FUNCTION_BLOCK SINGLE_EVENT_CONTROLLER (* Composite Function Block Type *)
  (* Standard: 61499-2 *)
  (* Version 1.0, 2019-03-16, adeel *)
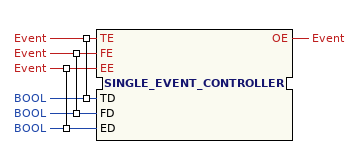
  EVENT_INPUT
    TE WITH TD; (* Initialization Request *)
    FE WITH FD; (* Normal Execution Request *)
    EE WITH ED;
  END_EVENT
  EVENT_OUTPUT
    OE; (* Initialization Confirm *)
  END_EVENT
  VAR_INPUT
    TD : BOOL; (* Input event qualifier *)
    FD : BOOL;
    ED : BOOL;
  END_VAR
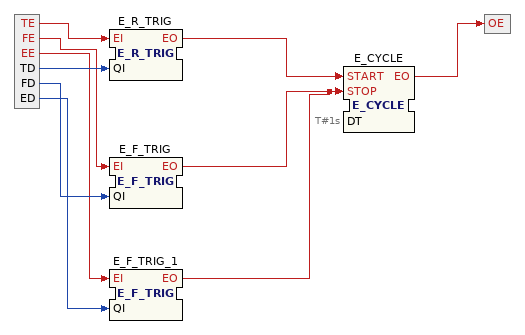
  FBS
    E_CYCLE : E_CYCLE(DT := T#1s);
    E_R_TRIG : E_R_TRIG;
    E_F_TRIG : E_F_TRIG;
    E_F_TRIG_1 : E_F_TRIG;
  END_FBS
  EVENT_CONNECTIONS
    E_R_TRIG.EO TO E_CYCLE.START;
    E_F_TRIG.EO TO E_CYCLE.STOP;
    TE TO E_R_TRIG.EI;
    FE TO E_F_TRIG.EI;
    E_CYCLE.EO TO OE;
    EE TO E_F_TRIG_1.EI;
    E_F_TRIG_1.EO TO E_CYCLE.STOP;
  END_CONNECTIONS
  DATA_CONNECTIONS
    TD TO E_R_TRIG.QI;
    FD TO E_F_TRIG.QI;
    ED TO E_F_TRIG_1.QI;
  END_CONNECTIONS
END_FUNCTION_BLOCK
